# EPICS autosave request: pointGreyApp/Db/pointGreyPropertyAbs_settings.req
$(P)$(R)$(PROPERTY)ValAbs
$(P)$(R)$(PROPERTY)AutoMode
